// TIA Portal project "box sorting" (V16)
// Vorlageprojekt für das Buch mit Zielsystem S7-1200

(* hardware
DEVICE "S7-1200-Station_1"  S7-1200 Station
   slot 0: "Baugruppenträger_0"  Rack  V1.0
   slot 1: "PLC_1"  CPU 1211C DC/DC/DC  6ES7 211-1AE40-0XB0  V4.1
*)

// ===== PLC "PLC_1"  CPU 1211C DC/DC/DC =====

VAR_GLOBAL   // PLC tag table "Standard-Variablentabelle"
   "start" AT %I0.0 : Bool;
   "primary conv" AT %Q0.0 : Bool;
   "sorting arm" AT %Q0.1 : Bool;
   "alarm" AT %Q0.2 : Bool;
   "low" AT %I0.1 : Bool;
   "up" AT %I0.2 : Bool;
   "low mtag" AT %M0.1 : Bool;
   "ctu down tag" AT %M0.2 : Bool;
   "up mtag" AT %M0.3 : Bool;
   "ctu up tag" AT %M0.4 : Bool;
END_VAR

// folder: System blocks/Program resources

DATA_BLOCK "IEC_Counter_0_DB_1"   // DB3
{ S7_Optimized_Access := 'TRUE' }
AUTHOR : Simatic
FAMILY : IEC
NAME : CNTR
VERSION : 1.0
// stored: InstanceOfName IEC_COUNTER
"IEC_COUNTER"
BEGIN
END_DATA_BLOCK

DATA_BLOCK "IEC_Counter_0_DB_2"   // DB4
{ S7_Optimized_Access := 'TRUE' }
AUTHOR : Simatic
FAMILY : IEC
NAME : CNTR
VERSION : 1.0
// stored: InstanceOfName IEC_COUNTER
"IEC_COUNTER"
BEGIN
END_DATA_BLOCK

DATA_BLOCK "IEC_Timer_0_DB"   // DB5
{ S7_Optimized_Access := 'TRUE' }
AUTHOR : Simatic
FAMILY : IEC
NAME : IEC_TMR
VERSION : 1.0
// stored: InstanceOfName IEC_TIMER
"IEC_TIMER"
BEGIN
END_DATA_BLOCK

DATA_BLOCK "IEC_Timer_0_DB_1"   // DB7
{ S7_Optimized_Access := 'TRUE' }
AUTHOR : Simatic
FAMILY : IEC
NAME : IEC_TMR
VERSION : 1.0
// stored: InstanceOfName IEC_TIMER
"IEC_TIMER"
BEGIN
END_DATA_BLOCK

// folder: (top level)

FUNCTION "MHJ-PLC-Lab-Function-S71200" : Void   // FC9000, SCL
{ S7_Optimized_Access := 'TRUE' }
VERSION : 0.1
   VAR_TEMP
      rdTimeReturn : Int;
      outputTime : DTL;
      SyncVal : Byte;
      forVal : Int;
      forVal_2 : Int;
      Value : Byte;
   END_VAR
   VAR CONSTANT
      CompVal : Byte := 16#34;
      Value_01 : Byte := 16#11;
      Value_01_DW : DWord := 16#A165_D992;
      Value_02_DW : DWord := 16#58BE_4401;
   END_VAR
BEGIN

   #Value:=PEEK(area := 16#82,
        dbNumber := 0,
        byteOffset := 511);
   #Value := #Value + 1;

   POKE(area := 16#82,
        dbNumber := 0,
        byteOffset := 511,
        value := #Value);

   POKE(area:=16#81,
        dbNumber:=0,
        byteOffset:=1016,
        value:=#Value_01_DW);
   POKE(area := 16#81,
        dbNumber := 0,
        byteOffset := 1020,
        value := #Value_02_DW);

   POKE(area := 16#81,
        dbNumber := 0,
        byteOffset := 511,
        value := B#16#00);

   FOR #forVal := 0 TO 120 DO
       FOR #forVal_2:=0 TO 10 DO
           #rdTimeReturn:=RD_SYS_T(#outputTime);
           #rdTimeReturn := WR_SYS_T(#outputTime);
           #rdTimeReturn := RD_SYS_T(#outputTime);
           #rdTimeReturn := WR_SYS_T(#outputTime);
       END_FOR;
       #SyncVal:= PEEK(area := 16#81,
                      dbNumber := 0,
                      byteOffset := 511);
       IF #SyncVal = #CompVal THEN
          GOTO M_1;
       END_IF;
   END_FOR;
   RETURN;

   M_1:
   POKE(area := 16#81,
        dbNumber := 0,
        byteOffset := 511,
        value := B#16#0);
END_FUNCTION

ORGANIZATION_BLOCK "Main"   // OB1, LAD, ProgramCycle
TITLE = "Main Program Sweep (Cycle)"
{ S7_Optimized_Access := 'TRUE' }
VERSION : 0.1
   VAR_INPUT
      Initial_Call : Bool;   // Initial call of this OB
      Remanence : Bool;   // =True, if remanent data are available
   END_VAR
   VAR_TEMP   // added for the SCL form of the ladder/FBD networks
      _w1 : Bool;
   END_VAR
BEGIN

REGION Network 1: Konnektierungsbaustein für PLC-Lab
   // Im Netzwerk 1 wird der Konnektierungsbaustein für PLC-Lab aufgerufen.
   // Dieser Aufruf darf nicht entfernt werden!
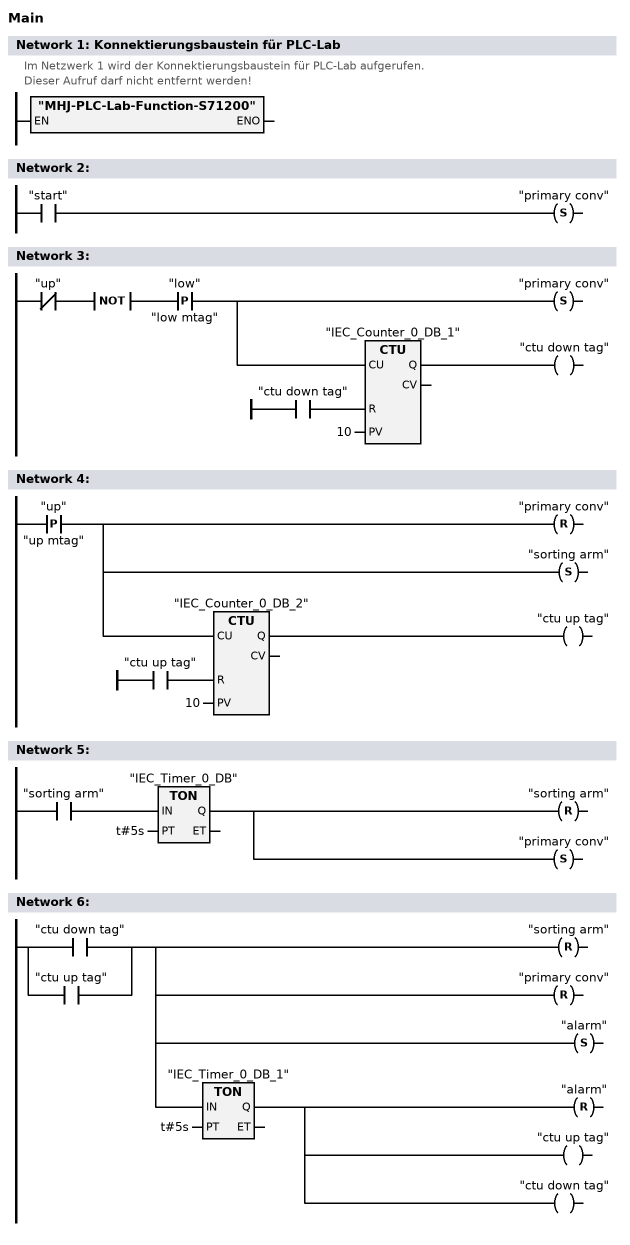
   RUNG wire#powerrail
      "MHJ-PLC-Lab-Function-S71200"()
   END_RUNG
   // the same network as SCL:
   "MHJ-PLC-Lab-Function-S71200"();
END_REGION

REGION Network 2
   RUNG wire#powerrail
      Contact( "start" )
      S_Coil( "primary conv" )
   END_RUNG
   // the same network as SCL:
   IF "start" THEN "primary conv" := TRUE; END_IF;
END_REGION

REGION Network 3
   #_w1 := NOT (NOT "up") AND "low" AND NOT "low mtag";   // rising edge of "low"
   "low mtag" := "low";
   IF #_w1 THEN "primary conv" := TRUE; END_IF;
   "IEC_Counter_0_DB_1".CTU(CU := #_w1, R := "ctu down tag", PV := 10);
   "ctu down tag" := "IEC_Counter_0_DB_1".Q;
END_REGION

REGION Network 4
   #_w1 := "up" AND NOT "up mtag";   // rising edge of "up"
   "up mtag" := "up";
   IF #_w1 THEN
       "primary conv" := FALSE;
       "sorting arm" := TRUE;
   END_IF;
   "IEC_Counter_0_DB_2".CTU(CU := #_w1, R := "ctu up tag", PV := 10);
   "ctu up tag" := "IEC_Counter_0_DB_2".Q;
END_REGION

REGION Network 5
   "IEC_Timer_0_DB".TON(IN := "sorting arm", PT := t#5s);
   IF "IEC_Timer_0_DB".Q THEN
       "sorting arm" := FALSE;
       "primary conv" := TRUE;
   END_IF;
END_REGION

REGION Network 6
   #_w1 := "ctu down tag" OR "ctu up tag";
   IF #_w1 THEN
       "sorting arm" := FALSE;
       "primary conv" := FALSE;
       "alarm" := TRUE;
   END_IF;
   "IEC_Timer_0_DB_1".TON(IN := #_w1, PT := t#5s);
   IF "IEC_Timer_0_DB_1".Q THEN "alarm" := FALSE; END_IF;
   "ctu up tag" := "IEC_Timer_0_DB_1".Q;
   "ctu down tag" := "IEC_Timer_0_DB_1".Q;
END_REGION
END_ORGANIZATION_BLOCK